Fanuc KAREL source: kb00061.KL

PROGRAM KB00061
%NOLOCKGROUP
%ENVIRONMENT FDEV
VAR
P1 : STRING[80];P2:BOOLEAN;P3:INTEGER
BEGIN
--
--
P1='A'
P2=TRUE
P3=1
DELETE_FILE(P1,P2,P3)
END KB00061
